FUNCTION_BLOCK FB_NestTableManager
VAR
    aNestInternal           : ARRAY[1..4] OF ST_Nest;
    aNestStatisticsInternal : ARRAY[1..4] OF ST_NestStatistics;
    aPositionToNest         : ARRAY[1..4] OF UINT := [1,2,3,4];
    bInitialised            : BOOL;
    i                       : INT;
    uiNest                  : UINT;
    uiMethodNestId          : UINT;
	bStatisticsEvent        : BOOL := FALSE;
	uiStatisticsEventNestId : UINT := 0;
	bStatisticsEventPassed  : BOOL := FALSE;
END_VAR

METHOD PUBLIC ClearOperatorNest
VAR_INPUT ePosition : E_TablePosition; END_VAR
uiMethodNestId := GetNestIdAtPosition(ePosition);

IF uiMethodNestId >= 1 AND uiMethodNestId <= 4 THEN
    aNestInternal[uiMethodNestId].bPbupPresent := FALSE;
    aNestInternal[uiMethodNestId].bLoadSetComplete := FALSE;
    aNestInternal[uiMethodNestId].bProcessRequired := FALSE;
    aNestInternal[uiMethodNestId].bProcessComplete := FALSE;
    aNestInternal[uiMethodNestId].eDisposition := E_PartDisposition.None;
    aNestInternal[uiMethodNestId].bDispositionSent := FALSE;
    aNestInternal[uiMethodNestId].bOperatorExchangeComplete := FALSE;

    aNestInternal[uiMethodNestId].stPatchDispenseResult.bValid := FALSE;
    aNestInternal[uiMethodNestId].stPatchDispenseResult.bPassed := FALSE;
    aNestInternal[uiMethodNestId].stPatchDispenseResult.eCode := E_ProcessResultCode.None;
    aNestInternal[uiMethodNestId].stHeatStakeResult.bValid := FALSE;
    aNestInternal[uiMethodNestId].stHeatStakeResult.bPassed := FALSE;
    aNestInternal[uiMethodNestId].stHeatStakeResult.eCode := E_ProcessResultCode.None;
    aNestInternal[uiMethodNestId].stVisionResult.bValid := FALSE;
    aNestInternal[uiMethodNestId].stVisionResult.bPassed := FALSE;
    aNestInternal[uiMethodNestId].stVisionResult.eCode := E_ProcessResultCode.None;

    aNestInternal[uiMethodNestId].ePatchDispenseStage := E_NestStageStatus.Waiting;
    aNestInternal[uiMethodNestId].eHeatStakeStage := E_NestStageStatus.Waiting;
    aNestInternal[uiMethodNestId].eVisionStage := E_NestStageStatus.Waiting;

    aNestInternal[uiMethodNestId].stResult.bValid := FALSE;
    aNestInternal[uiMethodNestId].stResult.bPassed := FALSE;
    aNestInternal[uiMethodNestId].stResult.eCode := E_ProcessResultCode.None;
    aNestInternal[uiMethodNestId].bStatisticsCounted := FALSE;
END_IF
END_METHOD

METHOD PUBLIC Cyclic
VAR_INPUT
    bIndexStable : BOOL;
    eIndexPosition : E_TablePosition;
    eOperatorPosition : E_TablePosition;
    bPartPresent : BOOL;
    bPbupPresent : BOOL;
    bOperatorReloadPermitted : BOOL;
    aNestEnabled : ARRAY[1..4] OF BOOL;
END_VAR
VAR
    bOperatorRecordProtected : BOOL;
END_VAR
IF NOT bInitialised THEN
    FOR i := 1 TO 4 DO
        aNestInternal[i].nId := INT_TO_UINT(i);
        aNestStatisticsInternal[i].uiNestId := INT_TO_UINT(i);
    END_FOR
    bInitialised := TRUE;
END_IF
FOR i := 1 TO 4 DO
    aNestInternal[i].bEnabled := aNestEnabled[i];
    // Pulse semantics do not depend on whether the index is moving.
    aNestInternal[i].bPartLoadedPulse := FALSE;
    aNestInternal[i].bPartRemovedPulse := FALSE;
END_FOR
IF bIndexStable AND (eIndexPosition <> E_TablePosition.Unknown) THEN
    CASE eIndexPosition OF
        E_TablePosition.Position1:
            aPositionToNest[1] := 1;
            aPositionToNest[2] := 4;
            aPositionToNest[3] := 3;
            aPositionToNest[4] := 2;
        E_TablePosition.Position2:
            aPositionToNest[1] := 2;
            aPositionToNest[2] := 1;
            aPositionToNest[3] := 4;
            aPositionToNest[4] := 3;
        E_TablePosition.Position3:
            aPositionToNest[1] := 3;
            aPositionToNest[2] := 2;
            aPositionToNest[3] := 1;
            aPositionToNest[4] := 4;
        E_TablePosition.Position4:
            aPositionToNest[1] := 4;
            aPositionToNest[2] := 3;
            aPositionToNest[3] := 2;
            aPositionToNest[4] := 1;
    END_CASE
    FOR i := 1 TO 4 DO
        aNestInternal[aPositionToNest[i]].ePosition := UINT_TO_E_TablePosition(INT_TO_UINT(i));
        aNestInternal[i].bPartLoadedPulse := FALSE;
        aNestInternal[i].bPartRemovedPulse := FALSE;
    END_FOR
    uiNest := aPositionToNest[TO_UINT(eOperatorPosition)];
    // Preserve a completed/reprocess product while its operator/reject exchange is pending.
    bOperatorRecordProtected := aNestInternal[uiNest].stResult.bValid
        OR (aNestInternal[uiNest].eDisposition = E_PartDisposition.Reprocess);
    aNestInternal[uiNest].bPartLoadedPulse := bPartPresent
        AND ((NOT bOperatorRecordProtected AND NOT aNestInternal[uiNest].bPreviousPartPresent)
            OR (bOperatorRecordProtected AND bOperatorReloadPermitted));

    aNestInternal[uiNest].bPartRemovedPulse :=
        NOT bPartPresent AND aNestInternal[uiNest].bPreviousPartPresent;

    IF aNestInternal[uiNest].bPartLoadedPulse THEN
        aNestInternal[uiNest].bProcessRequired := TRUE;
        aNestInternal[uiNest].bProcessComplete := FALSE;
        aNestInternal[uiNest].eDisposition := E_PartDisposition.None;
        aNestInternal[uiNest].bDispositionSent := FALSE;
        aNestInternal[uiNest].bOperatorExchangeComplete := FALSE;

        aNestInternal[uiNest].stPatchDispenseResult.bValid := FALSE;
        aNestInternal[uiNest].stPatchDispenseResult.bPassed := FALSE;
        aNestInternal[uiNest].stPatchDispenseResult.eCode := E_ProcessResultCode.None;
        aNestInternal[uiNest].stHeatStakeResult.bValid := FALSE;
        aNestInternal[uiNest].stHeatStakeResult.bPassed := FALSE;
        aNestInternal[uiNest].stHeatStakeResult.eCode := E_ProcessResultCode.None;
        aNestInternal[uiNest].stVisionResult.bValid := FALSE;
        aNestInternal[uiNest].stVisionResult.bPassed := FALSE;
        aNestInternal[uiNest].stVisionResult.eCode := E_ProcessResultCode.None;

        aNestInternal[uiNest].ePatchDispenseStage := E_NestStageStatus.Waiting;
        aNestInternal[uiNest].eHeatStakeStage := E_NestStageStatus.Waiting;
        aNestInternal[uiNest].eVisionStage := E_NestStageStatus.Waiting;

        aNestInternal[uiNest].stResult.bValid := FALSE;
        aNestInternal[uiNest].stResult.bPassed := FALSE;
        aNestInternal[uiNest].stResult.eCode := E_ProcessResultCode.None;
        aNestInternal[uiNest].bStatisticsCounted := FALSE;
    END_IF

    // Raw PBUP pocket presence is current at Operator, frozen while the nest travels.
    aNestInternal[uiNest].bPbupPresent := bPbupPresent;
    // A PBUP assembled at Vision may no longer occupy its original pocket.
    // Do not overwrite the paired-load history of a returned processed product.
    IF NOT bOperatorRecordProtected OR aNestInternal[uiNest].bPartLoadedPulse THEN
        aNestInternal[uiNest].bLoadSetComplete := bPartPresent AND bPbupPresent;
    END_IF
    aNestInternal[uiNest].bPreviousPartPresent := bPartPresent;
    aNestInternal[uiNest].bPartPresent := bPartPresent;
END_IF
END_METHOD

METHOD PUBLIC FinaliseResultAtPosition : BOOL
VAR_INPUT
    ePosition : E_TablePosition;
END_VAR
VAR
    uiId : UINT;
END_VAR

FinaliseResultAtPosition := FALSE;
uiId := GetNestIdAtPosition(ePosition);

IF (uiId >= 1) AND (uiId <= 4) THEN

    // =====================================================
    // REPROCESS PROTECTION
    // =====================================================
    // Reprocess is not a definitive product result.
    // Never convert it to Pass or Reject.
    // Never increment statistics for this attempt.

    IF aNestInternal[uiId].eDisposition = E_PartDisposition.Reprocess THEN
        RETURN;
    END_IF

    // No part in this physical nest: there is no product result to finalise.
    // No part in this physical nest: there is no product result to finalise.
    IF NOT aNestInternal[uiId].bPartPresent THEN

        aNestInternal[uiId].stResult.bValid := FALSE;
        aNestInternal[uiId].stResult.bPassed := FALSE;
        aNestInternal[uiId].stResult.eCode := E_ProcessResultCode.None;

        aNestInternal[uiId].bProcessComplete := TRUE;
        aNestInternal[uiId].bProcessRequired := FALSE;

        FinaliseResultAtPosition := TRUE;

    // A product result can only be finalised after all three process stages
    // have left Waiting.
    ELSIF
        (aNestInternal[uiId].ePatchDispenseStage <> E_NestStageStatus.Waiting)
        AND (aNestInternal[uiId].eHeatStakeStage <> E_NestStageStatus.Waiting)
        AND (aNestInternal[uiId].eVisionStage <> E_NestStageStatus.Waiting)
    THEN

        aNestInternal[uiId].stResult.bValid := TRUE;

        // =====================================================
        // FINAL PRODUCT RESULT
        // =====================================================
        // PASS is only possible when ALL three required
        // PatchPress processes have individually passed.
        //
        // Any other completed combination is a final FAIL,
        // including combinations containing NotTested.
        //
        // Examples:
        // Pass + Pass + Pass           -> PASS
        // Pass + Pass + Fail           -> FAIL
        // Pass + Fail + NotTested      -> FAIL
        // Fail + NotTested + NotTested -> FAIL
        // Pass + NotTested + NotTested -> FAIL

		IF
			(aNestInternal[uiId].ePatchDispenseStage = E_NestStageStatus.Complete)
			AND (aNestInternal[uiId].eHeatStakeStage = E_NestStageStatus.Complete)
			AND (aNestInternal[uiId].eVisionStage = E_NestStageStatus.Complete)
		THEN

            aNestInternal[uiId].stResult.bPassed := TRUE;
            aNestInternal[uiId].stResult.eCode := E_ProcessResultCode.Pass;
            aNestInternal[uiId].eDisposition := E_PartDisposition.Pass;
            aNestInternal[uiId].stResult.sDetail :=
                'Patch Press final result: PASS';

        ELSE

            aNestInternal[uiId].stResult.bPassed := FALSE;
            aNestInternal[uiId].stResult.eCode := E_ProcessResultCode.Fail;
            aNestInternal[uiId].eDisposition := E_PartDisposition.Reject;
            aNestInternal[uiId].stResult.sDetail :=
                'Patch Press final result: FAIL';

        END_IF

        aNestInternal[uiId].bProcessComplete := TRUE;
        aNestInternal[uiId].bProcessRequired := FALSE;

        // =====================================================
        // PRODUCTION STATISTICS
        // =====================================================
        // Count the final product result exactly once for this
        // physical nest.
        IF NOT aNestInternal[uiId].bStatisticsCounted THEN

            aNestStatisticsInternal[uiId].udiTotalTests :=
                aNestStatisticsInternal[uiId].udiTotalTests + 1;

            IF aNestInternal[uiId].stResult.bPassed THEN

                aNestStatisticsInternal[uiId].udiGoodParts :=
                    aNestStatisticsInternal[uiId].udiGoodParts + 1;

            ELSE

                aNestStatisticsInternal[uiId].udiBadParts :=
                    aNestStatisticsInternal[uiId].udiBadParts + 1;

            END_IF

            IF aNestStatisticsInternal[uiId].udiTotalTests > 0 THEN

                aNestStatisticsInternal[uiId].lrEfficiency :=
                    UDINT_TO_LREAL(
                        aNestStatisticsInternal[uiId].udiGoodParts
                    )
                    * 100.0
                    / UDINT_TO_LREAL(
                        aNestStatisticsInternal[uiId].udiTotalTests
                    );

            ELSE

                aNestStatisticsInternal[uiId].lrEfficiency := 0.0;

            END_IF
			
			// Generate a one-shot event when this product is counted.
			// The machine uses this event to create exactly one
			// Test History entry for the completed product.
			bStatisticsEvent := TRUE;
			uiStatisticsEventNestId := uiId;
			bStatisticsEventPassed := aNestInternal[uiId].stResult.bPassed;
            aNestInternal[uiId].bStatisticsCounted := TRUE;

        END_IF

        FinaliseResultAtPosition := TRUE;

    END_IF

END_IF
END_METHOD

METHOD PUBLIC GetAllNests : ARRAY[1..4] OF ST_Nest
GetAllNests := aNestInternal;
END_METHOD

METHOD PUBLIC GetAllNestStatistics : ARRAY[1..4] OF ST_NestStatistics
GetAllNestStatistics := aNestStatisticsInternal;
END_METHOD

METHOD PUBLIC GetNestAtPosition : ST_Nest
VAR_INPUT ePosition : E_TablePosition; END_VAR
uiMethodNestId := GetNestIdAtPosition(ePosition); IF uiMethodNestId >= 1 AND uiMethodNestId <= 4 THEN GetNestAtPosition := aNestInternal[uiMethodNestId]; END_IF
END_METHOD

METHOD PUBLIC GetNestIdAtPosition : UINT
VAR_INPUT ePosition : E_TablePosition; END_VAR
IF ePosition >= E_TablePosition.Position1 AND ePosition <= E_TablePosition.Position4 THEN GetNestIdAtPosition := aPositionToNest[TO_UINT(ePosition)]; ELSE GetNestIdAtPosition := 0; END_IF
END_METHOD

METHOD PUBLIC MarkHeatStakeNotTestedAtPosition
VAR_INPUT ePosition : E_TablePosition; END_VAR
VAR uiId : UINT; END_VAR

uiId := GetNestIdAtPosition(ePosition);
IF (uiId >= 1) AND (uiId <= 4) THEN
    IF aNestInternal[uiId].eHeatStakeStage <> E_NestStageStatus.Waiting THEN
        RETURN;
    END_IF
    aNestInternal[uiId].stHeatStakeResult.bValid := FALSE;
    aNestInternal[uiId].stHeatStakeResult.bPassed := FALSE;
    aNestInternal[uiId].stHeatStakeResult.eCode := E_ProcessResultCode.None;
    aNestInternal[uiId].eHeatStakeStage := E_NestStageStatus.NotTested;
END_IF
END_METHOD

METHOD PUBLIC MarkPatchDispenseNotTestedAtPosition
VAR_INPUT ePosition : E_TablePosition; END_VAR
VAR uiId : UINT; END_VAR

uiId := GetNestIdAtPosition(ePosition);
IF (uiId >= 1) AND (uiId <= 4) THEN
    IF aNestInternal[uiId].ePatchDispenseStage <> E_NestStageStatus.Waiting THEN
        RETURN;
    END_IF
    aNestInternal[uiId].stPatchDispenseResult.bValid := FALSE;
    aNestInternal[uiId].stPatchDispenseResult.bPassed := FALSE;
    aNestInternal[uiId].stPatchDispenseResult.eCode := E_ProcessResultCode.None;
    aNestInternal[uiId].ePatchDispenseStage := E_NestStageStatus.NotTested;
END_IF
END_METHOD

METHOD PUBLIC MarkReprocessAtPosition : BOOL
VAR_INPUT
    ePosition : E_TablePosition;
END_VAR
VAR
    uiId : UINT;
END_VAR
MarkReprocessAtPosition := FALSE;

uiId := GetNestIdAtPosition(ePosition);

IF (uiId >= 1) AND (uiId <= 4) THEN

    IF aNestInternal[uiId].bPartPresent THEN

        // -------------------------------------------------
        // PART DISPOSITION
        // -------------------------------------------------
        // The part did not complete the production process.
        // It must be removed by the operator and may be
        // reintroduced later as a completely new part.
        aNestInternal[uiId].eDisposition :=
            E_PartDisposition.Reprocess;

        // -------------------------------------------------
        // FINAL PRODUCT RESULT
        // -------------------------------------------------
        // Reprocess is deliberately NOT a final PASS/FAIL.
        // Therefore the final product result remains invalid.
        //
        // This prevents:
        // - Good Parts increment
        // - Bad Parts increment
        // - Test History entry
        aNestInternal[uiId].stResult.bValid := FALSE;
        aNestInternal[uiId].stResult.bPassed := FALSE;
        aNestInternal[uiId].stResult.eCode :=
            E_ProcessResultCode.None;

        // -------------------------------------------------
        // PROCESS CONTROL
        // -------------------------------------------------
        // No further production process shall be requested
        // for this part. It must travel directly through the
        // remaining stations until it reaches the operator.
        aNestInternal[uiId].bProcessRequired := FALSE;
        aNestInternal[uiId].bProcessComplete := TRUE;

        // -------------------------------------------------
        // STATISTICS
        // -------------------------------------------------
        // A Reprocess part is neither Good nor Bad.
        // No production counter is incremented here.
        aNestInternal[uiId].bStatisticsCounted := FALSE;

        MarkReprocessAtPosition := TRUE;

    END_IF

END_IF
END_METHOD

METHOD PUBLIC MarkVisionNotTestedAtPosition
VAR_INPUT ePosition : E_TablePosition; END_VAR
VAR uiId : UINT; END_VAR

uiId := GetNestIdAtPosition(ePosition);
IF (uiId >= 1) AND (uiId <= 4) THEN
    IF aNestInternal[uiId].eVisionStage <> E_NestStageStatus.Waiting THEN
        RETURN;
    END_IF
    aNestInternal[uiId].stVisionResult.bValid := FALSE;
    aNestInternal[uiId].stVisionResult.bPassed := FALSE;
    aNestInternal[uiId].stVisionResult.eCode := E_ProcessResultCode.None;
    aNestInternal[uiId].eVisionStage := E_NestStageStatus.NotTested;
END_IF
END_METHOD

METHOD PUBLIC ResetNestStatistics
VAR_INPUT
    uiNestId : UINT;
END_VAR
// =====================================================
// RESET NEST PRODUCTION STATISTICS
// =====================================================
// Reset only the accumulated production counters for
// the selected physical nest.
//
// IMPORTANT:
// - Test History is preserved.
// - Current nest/process results are preserved.
// - Part presence is preserved.
// - bStatisticsCounted is preserved so that a product
//   already counted before the reset cannot be counted
//   again simply because the statistics were cleared.

IF (uiNestId >= 1) AND (uiNestId <= 4) THEN

    aNestStatisticsInternal[uiNestId].udiTotalTests := 0;
    aNestStatisticsInternal[uiNestId].udiGoodParts := 0;
    aNestStatisticsInternal[uiNestId].udiBadParts := 0;
    aNestStatisticsInternal[uiNestId].lrEfficiency := 0.0;

END_IF
END_METHOD

METHOD PUBLIC StoreHeatStakeResultAtPosition : BOOL
VAR_INPUT ePosition : E_TablePosition; stResult : ST_ProcessResult; END_VAR
VAR uiId : UINT; END_VAR

StoreHeatStakeResultAtPosition := FALSE;
uiId := GetNestIdAtPosition(ePosition);
IF uiId >= 1 AND uiId <= 4 THEN
    aNestInternal[uiId].stHeatStakeResult := stResult;
    IF stResult.bValid AND stResult.bPassed THEN
        aNestInternal[uiId].eHeatStakeStage := E_NestStageStatus.Complete;

    ELSIF stResult.bValid THEN
        // A Heat Stake failure makes Vision irrelevant for this part.
        aNestInternal[uiId].eHeatStakeStage := E_NestStageStatus.Fail;

        aNestInternal[uiId].stVisionResult.bValid := FALSE;
        aNestInternal[uiId].stVisionResult.bPassed := FALSE;
        aNestInternal[uiId].stVisionResult.eCode := E_ProcessResultCode.None;
        aNestInternal[uiId].eVisionStage := E_NestStageStatus.NotTested;
    END_IF

    StoreHeatStakeResultAtPosition := TRUE;
END_IF
END_METHOD

METHOD PUBLIC StorePatchDispenseResultAtPosition : BOOL
VAR_INPUT ePosition : E_TablePosition; stResult : ST_ProcessResult; END_VAR
VAR uiId : UINT; END_VAR

StorePatchDispenseResultAtPosition := FALSE;
uiId := GetNestIdAtPosition(ePosition);
IF uiId >= 1 AND uiId <= 4 THEN
    aNestInternal[uiId].stPatchDispenseResult := stResult;
    IF stResult.bValid AND stResult.bPassed THEN
        aNestInternal[uiId].ePatchDispenseStage := E_NestStageStatus.Complete;

    ELSIF stResult.bValid THEN
        // Patch Dispense is the first process station.
        // If it fails, continuing with Heat Stake or Vision would no longer
        // represent a valid product flow. The downstream stations are
        // therefore explicitly recorded as NotTested for this physical nest.
        aNestInternal[uiId].ePatchDispenseStage := E_NestStageStatus.Fail;

        aNestInternal[uiId].stHeatStakeResult.bValid := FALSE;
        aNestInternal[uiId].stHeatStakeResult.bPassed := FALSE;
        aNestInternal[uiId].stHeatStakeResult.eCode := E_ProcessResultCode.None;
        aNestInternal[uiId].eHeatStakeStage := E_NestStageStatus.NotTested;

        aNestInternal[uiId].stVisionResult.bValid := FALSE;
        aNestInternal[uiId].stVisionResult.bPassed := FALSE;
        aNestInternal[uiId].stVisionResult.eCode := E_ProcessResultCode.None;
        aNestInternal[uiId].eVisionStage := E_NestStageStatus.NotTested;
    END_IF

    StorePatchDispenseResultAtPosition := TRUE;
END_IF
END_METHOD

METHOD PUBLIC StoreVisionResultAtPosition : BOOL
VAR_INPUT ePosition : E_TablePosition; stResult : ST_ProcessResult; END_VAR
VAR uiId : UINT; END_VAR

StoreVisionResultAtPosition := FALSE;
uiId := GetNestIdAtPosition(ePosition);
IF uiId >= 1 AND uiId <= 4 THEN
    aNestInternal[uiId].stVisionResult := stResult;
    IF stResult.bValid AND stResult.bPassed THEN
        aNestInternal[uiId].eVisionStage := E_NestStageStatus.Complete;
    ELSIF stResult.bValid THEN
        aNestInternal[uiId].eVisionStage := E_NestStageStatus.Fail;
    END_IF
    StoreVisionResultAtPosition := TRUE;
END_IF
END_METHOD

END_FUNCTION_BLOCK

(* stored: Version 1.1.0.1, ProductVersion 3.1.4026.18
   POU FB_NestTableManager: Id {7d4da875-9776-4fb9-89ad-14daa86147a0}, SpecialFunc None
   Method ClearOperatorNest: Id {49a5db95-39d9-4d1e-a633-d63e9985b5f5}
   Method Cyclic: Id {5b54e275-1e8e-4728-a765-bebaee4a975e}
   Method FinaliseResultAtPosition: Id {103a97ef-17a2-465c-b799-3140c30b4be4}
   Method GetAllNests: Id {aa3853bc-758e-419d-be3c-5d9c11c9ea70}
   Method GetAllNestStatistics: Id {8b696e48-6e5b-41e1-b556-e697dd3d4800}
   Method GetNestAtPosition: Id {6f45a335-2486-4b63-8916-a95158ba88ea}
   Method GetNestIdAtPosition: Id {b88cece0-cb19-43ea-b8fc-aa98089534fa}
   Method MarkHeatStakeNotTestedAtPosition: Id {151c59e0-e047-4434-83b6-2583f0e0b1c0}
   Method MarkPatchDispenseNotTestedAtPosition: Id {a16e2a9e-2659-4648-bbbd-ab30e5fccc5c}
   Method MarkReprocessAtPosition: Id {11b84306-b654-4f16-a1e1-6ede3fcaa773}
   Method MarkVisionNotTestedAtPosition: Id {3fdd2071-dd2d-41d0-acd4-ba93bbfa2d17}
   Method ResetNestStatistics: Id {4686ed6c-445c-4fbb-85fb-9e3ed12abe11}
   Method StoreHeatStakeResultAtPosition: Id {47087ea7-1524-4d31-b8df-b5ffc8b33f8d}
   Method StorePatchDispenseResultAtPosition: Id {a92f119a-0c27-4512-8bbc-81ec3250a1f3}
   Method StoreVisionResultAtPosition: Id {be0b3a8a-2b1c-49f9-9df2-6bd47e39bcd4} *)
